(* IEC 61131-3 sources: axftcmlib/src/Guards, 3 files *)

(* ---- BinSignalRiseGuard.st ---- *)
USING Simatic.Ax.StateFramework;
USING Simatic.Ax.IO.Input;
NAMESPACE Simatic.Ax.axftcmlib

    CLASS BinSignalRiseGuard IMPLEMENTS IGuard
        VAR PUBLIC
           BinSignal : IBinSignal;
        END_VAR

        METHOD PUBLIC Check : BOOL
            Check := (BinSignal.QRis());
        END_METHOD

        METHOD PUBLIC Reset
            ;
        END_METHOD
    END_CLASS
END_NAMESPACE

(* ---- PLCOpentateGuard.st ---- *)
USING Simatic.Ax.StateFramework;
NAMESPACE Simatic.Ax.axftcmlib

    ///This guard is used to check the activity of an axis
    ///An Axis will return a PLCOpenSTate#Done if a movement is finished
    /// This is sed for state transitions
    CLASS PLCOpenstateGuard IMPLEMENTS IGuard
        VAR PUBLIC
            Axis : REF_TO Axis;
        END_VAR

        METHOD PUBLIC Check : BOOL
            Check := (Axis^.GetPlcOpenState() = PlcOpenState#Done);
        END_METHOD

        METHOD PUBLIC Reset
            ;
        END_METHOD
    END_CLASS
END_NAMESPACE

(* ---- StartGuard.st ---- *)
USING Simatic.Ax.StateFramework;

NAMESPACE Simatic.Ax.axftcmlib
    ///Guard used to start the actual statemachine
    /// Is used in the pneumatic cylinder class
    CLASS StartGuard IMPLEMENTS IGuard

        VAR
            IsStarted : BOOL;
        END_VAR

        METHOD PUBLIC Check : BOOL
            Check := IsStarted;
        END_METHOD

        METHOD PUBLIC Reset
            IsStarted := FALSE;
        END_METHOD

        METHOD PUBLIC Start
            IsStarted := TRUE;
        END_METHOD
    END_CLASS

END_NAMESPACE
